(* IEC 61131-3 sources: repolevel_ST_code_completion/output/0127完整版本_带planner/repoeval_plc_hello_mixing_tank/readful_result_history, 9 files *)

(* ---- F_ResetDeviceCommands_0.st ---- *)
FUNCTION F_ResetDeviceCommands : BOOL
VAR_IN_OUT
	// HMI命令标志（需要复位）
	bMixerRunCmd		:	BOOL;
	bMixerStopCmd		:	BOOL;
	bMedium1OpenCmd		:	BOOL;
	bMedium1CloseCmd	:	BOOL;
	bMedium2OpenCmd		:	BOOL;
	bMedium2CloseCmd	:	BOOL;
	bDrainOpenCmd		:	BOOL;
	bDrainCloseCmd		:	BOOL;
END_VAR
VAR_INPUT
	// 设备状态反馈
	bMixerRunning		:	BOOL;
	bMedium1Opened		:	BOOL;
	bMedium2Opened		:	BOOL;
	bDrainOpened		:	BOOL;
END_VAR
VAR
	bAllCommandsReset : BOOL := TRUE;
END_VAR

// 混合电机命令复位
IF bMixerRunning THEN
	bMixerRunCmd := FALSE;
	bMixerStopCmd := FALSE;
ELSE
	bAllCommandsReset := FALSE;
END_IF

// 介质1阀门命令复位
IF bMedium1Opened THEN
	bMedium1OpenCmd := FALSE;
	bMedium1CloseCmd := FALSE;
ELSE
	bAllCommandsReset := FALSE;
END_IF

// 介质2阀门命令复位
IF bMedium2Opened THEN
	bMedium2OpenCmd := FALSE;
	bMedium2CloseCmd := FALSE;
ELSE
	bAllCommandsReset := FALSE;
END_IF

// 排水阀门命令复位
IF bDrainOpened THEN
	bDrainOpenCmd := FALSE;
	bDrainCloseCmd := FALSE;
ELSE
	bAllCommandsReset := FALSE;
END_IF

// 返回所有命令是否已复位
F_ResetDeviceCommands := bAllCommandsReset;
RETURN;
END_FUNCTION

(* ---- F_UpdateLimitSwitches_0.st ---- *)
FUNCTION F_UpdateLimitSwitches : BOOL
VAR_INPUT
	rTankLevel			:	REAL;			// 当前液位 (%)
	rFullThreshold		:	REAL := 85.0;	// 满液位阈值 (%)
	rEmptyThreshold		:	REAL := 5.0;	// 空液位阈值 (%)
END_VAR
VAR_OUTPUT
	bLevelFull			:	BOOL;			// 液位满开关
	bLevelEmpty			:	BOOL;			// 液位空开关
END_VAR
bLevelFull := rTankLevel >= rFullThreshold;
bLevelEmpty := rTankLevel <= rEmptyThreshold;
F_UpdateLimitSwitches := TRUE;
RETURN;
END_FUNCTION

(* ---- FB_AutoSequence_0.st ---- *)
FUNCTION_BLOCK FB_AutoSequence
VAR_INPUT
	bEnable				:	BOOL;			// 使能自动序列
	bReset				:	BOOL;			// 复位到排空状态

	// 液位传感器反馈
	bTankLevelFull		:	BOOL;			// 液位满传感器
	bTankLevelEmpty		:	BOOL;			// 液位空传感器

	// 设备状态反馈
	bMixerRunning		:	BOOL;			// 混合电机运行中
	bMedium1Opened		:	BOOL;			// 介质1阀门打开
	bMedium2Opened		:	BOOL;			// 介质2阀门打开
	bDrainOpened		:	BOOL;			// 排空阀门打开

	// 配置参数
	tMixingDuration		:	TIME := T#10S;	// 混合持续时间
END_VAR
VAR_OUTPUT
	// 设备控制输出
	bMixerRunCmd		:	BOOL;			// 混合电机运行命令
	bMedium1OpenCmd		:	BOOL;			// 介质1阀门打开命令
	bMedium2OpenCmd		:	BOOL;			// 介质2阀门打开命令
	bDrainOpenCmd		:	BOOL;			// 排空阀门打开命令

	// 状态输出
	eCurrentState		:	AUTO_SEQUENCE;	// 当前状态
	nCyclesCompleted	:	UINT;			// 完成的循环次数
END_VAR
VAR
	tonMixing			:	TON;			// 混合定时器
END_VAR

// 初始化设备控制输出
bMixerRunCmd := FALSE;
bMedium1OpenCmd := FALSE;
bMedium2OpenCmd := FALSE;
bDrainOpenCmd := FALSE;

// 检查复位条件
IF bReset THEN
	eCurrentState := AUTO_SEQUENCE.DRAINING;
	nCyclesCompleted := 0;
	RETURN;
END_IF

// 检查使能条件
IF NOT bEnable THEN
	eCurrentState := AUTO_SEQUENCE.IDLE;
	RETURN;
END_IF

// 自动序列状态机
CASE eCurrentState OF
	AUTO_SEQUENCE.DRAINING:
		// 排空状态逻辑
		bDrainOpenCmd := TRUE;
		IF bTankLevelEmpty THEN
			eCurrentState := AUTO_SEQUENCE.FILLING;
		END_IF;

	AUTO_SEQUENCE.FILLING:
		// 填充状态逻辑
		bMedium1OpenCmd := TRUE;
		bMedium2OpenCmd := TRUE;
		IF bTankLevelFull THEN
			eCurrentState := AUTO_SEQUENCE.MIXING;
		END_IF;

	AUTO_SEQUENCE.MIXING:
		// 混合状态逻辑
		bMixerRunCmd := TRUE;
		tonMixing(IN := TRUE, PT := tMixingDuration);
		IF tonMixing.Q THEN
			eCurrentState := AUTO_SEQUENCE.DRAINING;
			nCyclesCompleted := nCyclesCompleted + 1;
		END_IF;

	ELSE
		// 默认状态为初始状态
		eCurrentState := AUTO_SEQUENCE.IDLE;
END_CASE
END_FUNCTION_BLOCK

(* ---- FB_AutoSequence_1.st ---- *)
FUNCTION_BLOCK FB_AutoSequence
VAR_INPUT
	bEnable				:	BOOL;			// 使能自动序列
	bReset				:	BOOL;			// 复位到排空状态

	// 液位传感器反馈
	bTankLevelFull		:	BOOL;			// 液位满传感器
	bTankLevelEmpty		:	BOOL;			// 液位空传感器

	// 设备状态反馈
	bMixerRunning		:	BOOL;			// 混合电机运行中
	bMedium1Opened		:	BOOL;			// 介质1阀门打开
	bMedium2Opened		:	BOOL;			// 介质2阀门打开
	bDrainOpened		:	BOOL;			// 排空阀门打开

	// 配置参数
	tMixingDuration		:	TIME := T#10S;	// 混合持续时间
END_VAR
VAR_OUTPUT
	// 设备控制输出
	bMixerRunCmd		:	BOOL;			// 混合电机运行命令
	bMedium1OpenCmd		:	BOOL;			// 介质1阀门打开命令
	bMedium2OpenCmd		:	BOOL;			// 介质2阀门打开命令
	bDrainOpenCmd		:	BOOL;			// 排空阀门打开命令

	// 状态输出
	eCurrentState		:	AUTO_SEQUENCE;	// 当前状态
	nCyclesCompleted	:	UINT;			// 完成的循环次数
END_VAR
VAR
	tonMixing			:	TON;			// 混合定时器
END_VAR

// 初始化设备控制输出
bMixerRunCmd := FALSE;
bMedium1OpenCmd := FALSE;
bMedium2OpenCmd := FALSE;
bDrainOpenCmd := FALSE;

// 检查复位条件
IF bReset THEN
// Replace AUTO_SEQUENCE.DRAINING with a constant value or default state
  eCurrentState := 0; // Assuming '0' corresponds to the DRAINING state
	nCyclesCompleted := 0;
	RETURN;
END_IF

// 检查使能条件
IF NOT bEnable THEN
// Replace AUTO_SEQUENCE.IDLE with a constant value or default state
  eCurrentState := 1; // Assuming '1' corresponds to the IDLE state
	RETURN;
END_IF

// 自动序列状态机
CASE eCurrentState OF
  0:	// DRAINING state
    // 排空状态逻辑
    bDrainOpenCmd := TRUE;
    IF bTankLevelEmpty THEN
      eCurrentState := 2; // Transition to FILLING state
    END_IF;

  2:	// FILLING state
    // 填充状态逻辑
    bMedium1OpenCmd := TRUE;
    bMedium2OpenCmd := TRUE;
    IF bTankLevelFull THEN
      eCurrentState := 3; // Transition to MIXING state
    END_IF;

  3:	// MIXING state
    // 混合状态逻辑
    bMixerRunCmd := TRUE;
    tonMixing(IN := TRUE, PT := tMixingDuration);
    IF tonMixing.Q THEN
      eCurrentState := 0; // Transition back to DRAINING state
      nCyclesCompleted := nCyclesCompleted + 1;
    END_IF;

  ELSE
    // 默认状态为初始状态
    eCurrentState := 1; // IDLE state
END_CASE
END_FUNCTION_BLOCK

(* ---- FB_AutoSequence_2.st ---- *)
FUNCTION_BLOCK FB_AutoSequence
VAR_INPUT
	bEnable				:	BOOL;			// 使能自动序列
	bReset				:	BOOL;			// 复位到排空状态

	// 液位传感器反馈
	bTankLevelFull		:	BOOL;			// 液位满传感器
	bTankLevelEmpty		:	BOOL;			// 液位空传感器

	// 设备状态反馈
	bMixerRunning		:	BOOL;			// 混合电机运行中
	bMedium1Opened		:	BOOL;			// 介质1阀门打开
	bMedium2Opened		:	BOOL;			// 介质2阀门打开
	bDrainOpened		:	BOOL;			// 排空阀门打开

	// 配置参数
	tMixingDuration		:	TIME := T#10S;	// 混合持续时间
END_VAR
VAR_OUTPUT
	// 设备控制输出
	bMixerRunCmd		:	BOOL;			// 混合电机运行命令
	bMedium1OpenCmd		:	BOOL;			// 介质1阀门打开命令
	bMedium2OpenCmd		:	BOOL;			// 介质2阀门打开命令
	bDrainOpenCmd		:	BOOL;			// 排空阀门打开命令

	// 状态输出
	eCurrentState		:	AUTO_SEQUENCE;	// 当前状态
	nCyclesCompleted	:	UINT;			// 完成的循环次数
END_VAR
VAR
	tonMixing			:	TON;			// 混合定时器
END_VAR

// 初始化设备控制输出
bMixerRunCmd := FALSE;
bMedium1OpenCmd := FALSE;
bMedium2OpenCmd := FALSE;
bDrainOpenCmd := FALSE;

// 检查复位条件
IF bReset THEN
// Replace AUTO_SEQUENCE.DRAINING with a constant value or default state
  eCurrentState := 0; // Assuming '0' corresponds to the DRAINING state
	nCyclesCompleted := 0;
	RETURN;
END_IF

// 检查使能条件
IF NOT bEnable THEN
// Replace AUTO_SEQUENCE.IDLE with a constant value or default state
  eCurrentState := 1; // Assuming '1' corresponds to the IDLE state
	RETURN;
END_IF

// 自动序列状态机
CASE eCurrentState OF
 0:	// DRAINING state
  // 排空状态逻辑
  bDrainOpenCmd := TRUE;
  IF bTankLevelEmpty THEN
   eCurrentState := 2; // Transition to FILLING state
  END_IF;

 2:	// FILLING state
  // 填充状态逻辑
  bMedium1OpenCmd := TRUE;
  bMedium2OpenCmd := TRUE;
  IF bTankLevelFull THEN
   eCurrentState := 3; // Transition to MIXING state
  END_IF;

 3:	// MIXING state
  // 混合状态逻辑
  bMixerRunCmd := TRUE;
  tonMixing(IN := TRUE, PT := tMixingDuration);
  IF tonMixing.Q THEN
   eCurrentState := 0; // Transition back to DRAINING state
   nCyclesCompleted := nCyclesCompleted + 1;
  END_IF;

 ELSE
  // 默认状态为初始状态
  eCurrentState := 1; // IDLE state
END_CASE
END_FUNCTION_BLOCK

(* ---- FB_AutoSequence_3.st ---- *)
FUNCTION_BLOCK FB_AutoSequence
VAR_INPUT
	bEnable				:	BOOL;			// 使能自动序列
	bReset				:	BOOL;			// 复位到排空状态

	// 液位传感器反馈
	bTankLevelFull		:	BOOL;			// 液位满传感器
	bTankLevelEmpty		:	BOOL;			// 液位空传感器

	// 设备状态反馈
	bMixerRunning		:	BOOL;			// 混合电机运行中
	bMedium1Opened		:	BOOL;			// 介质1阀门打开
	bMedium2Opened		:	BOOL;			// 介质2阀门打开
	bDrainOpened		:	BOOL;			// 排空阀门打开

	// 配置参数
	tMixingDuration		:	TIME := T#10S;	// 混合持续时间
END_VAR
VAR_OUTPUT
	// 设备控制输出
	bMixerRunCmd		:	BOOL;			// 混合电机运行命令
	bMedium1OpenCmd		:	BOOL;			// 介质1阀门打开命令
	bMedium2OpenCmd		:	BOOL;			// 介质2阀门打开命令
	bDrainOpenCmd		:	BOOL;			// 排空阀门打开命令

	// 状态输出
	eCurrentState		:	AUTO_SEQUENCE;	// 当前状态
	nCyclesCompleted	:	UINT;			// 完成的循环次数
END_VAR
VAR
	tonMixing			:	TON;			// 混合定时器
END_VAR

// 初始化设备控制输出
bMixerRunCmd := FALSE;
bMedium1OpenCmd := FALSE;
bMedium2OpenCmd := FALSE;
bDrainOpenCmd := FALSE;

// 检查复位条件
IF bReset THEN
// Replace AUTO_SEQUENCE.DRAINING with a constant value or default state
  eCurrentState := 0; // Assuming '0' corresponds to the DRAINING state
	nCyclesCompleted := 0;
	RETURN;
END_IF

// 检查使能条件
IF NOT bEnable THEN
// Replace AUTO_SEQUENCE.IDLE with a constant value or default state
  eCurrentState := 1; // Assuming '1' corresponds to the IDLE state
	RETURN;
END_IF

// 自动序列状态机
CASE eCurrentState OF
0:	// DRAINING state
 // 排空状态逻辑
 bDrainOpenCmd := TRUE;
 IF bTankLevelEmpty THEN
 eCurrentState := 2; // Transition to FILLING state
 END_IF;

2:	// FILLING state
 // 填充状态逻辑
 bMedium1OpenCmd := TRUE;
 bMedium2OpenCmd := TRUE;
 IF bTankLevelFull THEN
 eCurrentState := 3; // Transition to MIXING state
 END_IF;

3:	// MIXING state
 // 混合状态逻辑
 bMixerRunCmd := TRUE;
 tonMixing(IN := TRUE, PT := tMixingDuration);
 IF tonMixing.Q THEN
 eCurrentState := 0; // Transition back to DRAINING state
 nCyclesCompleted := nCyclesCompleted + 1;
 END_IF;

ELSE
 // 默认状态为初始状态
 eCurrentState := 1; // IDLE state
END_CASE
END_FUNCTION_BLOCK

(* ---- FB_ManualControl_0.st ---- *)
FUNCTION_BLOCK FB_ManualControl
VAR_INPUT
	// HMI命令输入
	bMixerRunCmd		:	BOOL;
	bMixerStopCmd		:	BOOL;
	bMedium1OpenCmd		:	BOOL;
	bMedium1CloseCmd	:	BOOL;
	bMedium2OpenCmd		:	BOOL;
	bMedium2CloseCmd	:	BOOL;
	bDrainOpenCmd		:	BOOL;
	bDrainCloseCmd		:	BOOL;

	// 设备反馈输入
	bMixerRunning		:	BOOL;
	bMedium1Opened		:	BOOL;
	bMedium2Opened		:	BOOL;
	bDrainOpened		:	BOOL;
END_VAR
VAR_OUTPUT
	// 设备控制输出
	bMixerRunCmdOut		:	BOOL;
	bMedium1OpenCmdOut	:	BOOL;
	bMedium2OpenCmdOut	:	BOOL;
	bDrainOpenCmdOut	:	BOOL;
END_VAR
bMixerRunCmdOut := (bMixerRunCmd OR bMixerRunning) AND NOT bMixerStopCmd;

bMedium1OpenCmdOut := (bMedium1OpenCmd OR bMedium1Opened) AND NOT bMedium1CloseCmd;

bMedium2OpenCmdOut := (bMedium2OpenCmd OR bMedium2Opened) AND NOT bMedium2CloseCmd;

bDrainOpenCmdOut := (bDrainOpenCmd OR bDrainOpened) AND NOT bDrainCloseCmd;
END_FUNCTION_BLOCK

(* ---- FB_ModeController_0.st ---- *)
FUNCTION_BLOCK FB_ModeController
VAR_INPUT
	bSetToAuto		:	BOOL;	// 切换到自动模式命令
	bSetToManual	:	BOOL;	// 切换到手动模式命令
END_VAR
VAR_OUTPUT
	eCurrentMode	:	MODES;	// 当前模式
	bModeChanged	:	BOOL;	// 模式改变标志
END_VAR
VAR
	eLastMode		:	MODES;	// 上次模式
END_VAR

// 模式切换逻辑
IF bSetToAuto AND (eCurrentMode <> MODES.AUTO) THEN
	eCurrentMode := MODES.AUTO;
	bModeChanged := TRUE;
ELSIF bSetToManual AND (eCurrentMode <> MODES.MANUAL) THEN
	eCurrentMode := MODES.MANUAL;
	bModeChanged := TRUE;
ELSE
	bModeChanged := FALSE;
END_IF

// 更新上次模式
eLastMode := eCurrentMode;
END_FUNCTION_BLOCK

(* ---- FB_TankLevelSimulator_0.st ---- *)
FUNCTION_BLOCK FB_TankLevelSimulator
VAR_INPUT
	bMedium1Opened		:	BOOL;			// 介质1阀门打开
	bMedium2Opened		:	BOOL;			// 介质2阀门打开
	bDrainOpened		:	BOOL;			// 排空阀门打开
	bReset				:	BOOL;			// 复位到初始液位

	// 配置参数
	rInitialLevel		:	REAL := 25.0;	// 初始液位 (%)
	rFillRate1			:	REAL := 0.1;	// 介质1填充速率 (%/cycle)
	rFillRate2			:	REAL := 0.1;	// 介质2填充速率 (%/cycle)
	rDrainRate			:	REAL := 0.2;	// 排空速率 (%/cycle)
	rMinLevel			:	REAL := 0.0;	// 最小液位 (%)
	rMaxLevel			:	REAL := 100.0;	// 最大液位 (%)
END_VAR
VAR_OUTPUT
	rCurrentLevel		:	REAL;			// 当前液位 (%)
END_VAR
VAR
	rTempLevel : REAL; // 临时变量用于液位计算
END_VAR

// 复位逻辑
IF bReset THEN
	rCurrentLevel := rInitialLevel;
ELSE
	// 液位计算
	rTempLevel := rCurrentLevel
				+ rFillRate1 * BOOL_TO_REAL(bMedium1Opened)
				+ rFillRate2 * BOOL_TO_REAL(bMedium2Opened)
				- rDrainRate * BOOL_TO_REAL(bDrainOpened);

	// 边界检查
	IF rTempLevel > rMaxLevel THEN
		rCurrentLevel := rMaxLevel;
	ELSIF rTempLevel < rMinLevel THEN
		rCurrentLevel := rMinLevel;
	ELSE
		rCurrentLevel := rTempLevel;
	END_IF;
END_IF;
END_FUNCTION_BLOCK
